(* IEC 61131-3 sources: RL_MAR/experiments/comparison/autoplc/results/gpt-4o-mini_20260511_164212/med_73, 1 file *)

(* ---- med_73_3.st ---- *)
FUNCTION_BLOCK RoboticWeldingSystem
    VAR_INPUT
        RobotArm1Ready : BOOL; (* Input for robot arm 1 ready status *)
        RobotArm2Ready : BOOL; (* Input for robot arm 2 ready status *)
        WeldingGunReady : BOOL; (* Input for welding gun ready status *)
        StartButton : BOOL; (* Input for start button press *)
        StopButton : BOOL; (* Input for stop button press *)
    END_VAR

    VAR_OUTPUT
        WeldingTrigger : BOOL; (* Output to trigger welding *)
        WeldingComplete : BOOL; (* Output indicating welding completion *)
    END_VAR

    VAR
        State : INT; (* State variable to manage the control states *)
    END_VAR

    (* State Definitions *)
    CONST
        IDLE_STATE : INT := 0;
        WELDING_READY_STATE : INT := 1;
        WELDING_STATE : INT := 2;
        STOP_STATE : INT := 3;
    END_CONST

    (* Initialization *)
    IF State = IDLE_STATE THEN
        WeldingTrigger := FALSE;
        WeldingComplete := FALSE;
    END_IF

    (* State Evaluation *)
    CASE State OF
        IDLE_STATE:
            IF StopButton THEN
                WeldingTrigger := FALSE;
                WeldingComplete := TRUE;
                State := STOP_STATE;
            ELSIF RobotArm1Ready AND RobotArm2Ready AND WeldingGunReady AND StartButton THEN
                WeldingTrigger := TRUE;
                State := WELDING_READY_STATE;
            END_IF;

        WELDING_READY_STATE:
            IF StopButton THEN
                WeldingTrigger := FALSE;
                WeldingComplete := TRUE;
                State := STOP_STATE;
            ELSE
                State := WELDING_STATE; (* Transition to welding state *)
            END_IF;

        WELDING_STATE:
            IF StopButton THEN
                WeldingTrigger := FALSE;
                WeldingComplete := TRUE;
                State := STOP_STATE;
            ELSE
                (* Continue welding process *)
                WeldingComplete := FALSE; (* Welding is ongoing *)
            END_IF;

        STOP_STATE:
            (* In stop state, ensure welding is not triggered *)
            WeldingTrigger := FALSE;
            WeldingComplete := TRUE; (* Indicate welding is complete *)
            IF NOT StopButton THEN
                State := IDLE_STATE; (* Return to idle state if stop button is released *)
            END_IF;

    END_CASE;

END_FUNCTION_BLOCK
